(* PLC project Unnamed, Unknown Unnamed 1 *)
(* stored: creationDateTime 2024-11-21T00:40:53, modificationDateTime 2024-12-05T23:30:09 *)

(* LED *)
PROGRAM HelloWorld
  VAR
    Set : BOOL;
    Reset : BOOL;
    Hello_World : BOOL;
    Select : INT;
    Mode_1 : BOOL;
    Mode_2 : BOOL;
    Mode_3 : BOOL;
    Mode_4 : BOOL;
    LED : BOOL;
    LED0 : BOOL;
    R_TRIG0 : R_TRIG;
    F_TRIG0 : F_TRIG;
  END_VAR
  VAR  (* added by the conversion: wires and edge detectors of the diagram *)
    _MOVE27_ENO : BOOL;
    _MOVE27_OUT : INT;
  END_VAR

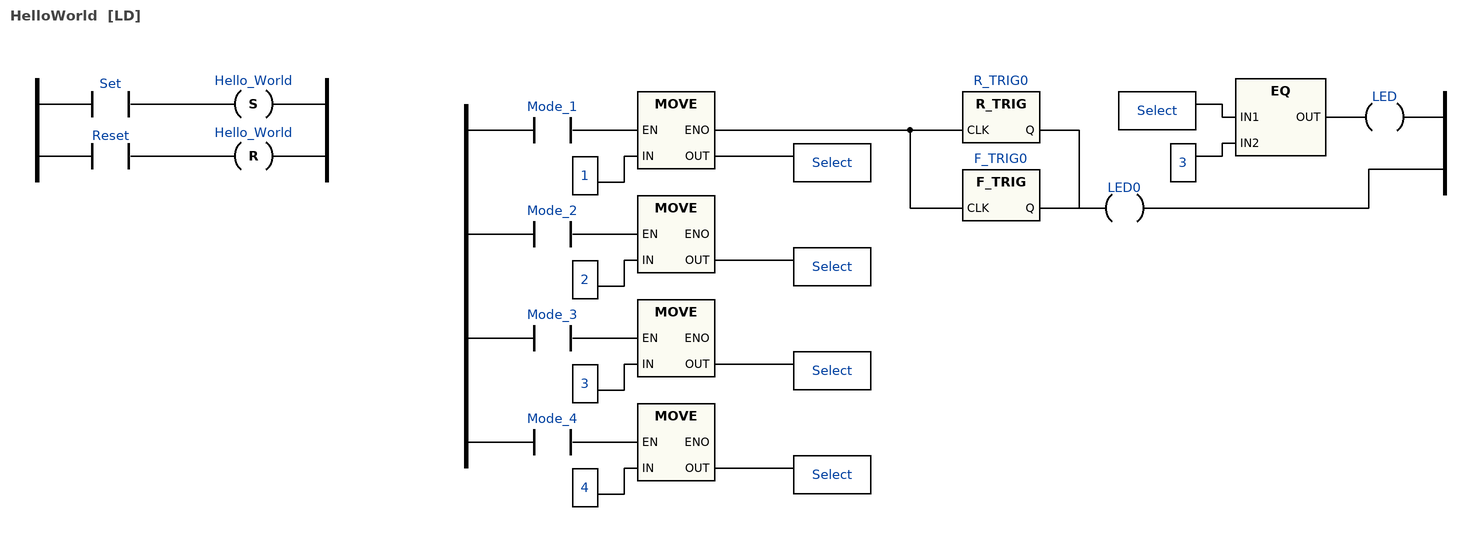
(* LD diagram, written out as Structured Text *)
IF Set THEN Hello_World := TRUE; END_IF;
IF Reset THEN Hello_World := FALSE; END_IF;
_MOVE27_OUT := MOVE(EN := Mode_1, IN := 1, ENO => _MOVE27_ENO);
IF _MOVE27_ENO THEN Select := _MOVE27_OUT; END_IF;
IF Mode_2 THEN Select := 2; END_IF;
IF Mode_3 THEN Select := 3; END_IF;
IF Mode_4 THEN Select := 4; END_IF;
LED := Select = 3;
R_TRIG0(CLK := _MOVE27_ENO);
F_TRIG0(CLK := _MOVE27_ENO);
LED0 := R_TRIG0.Q OR F_TRIG0.Q;
END_PROGRAM

CONFIGURATION Config0
  RESOURCE Res0 ON PLC
    TASK task0(INTERVAL := T#20ms, PRIORITY := 0);
    PROGRAM instance0 WITH task0 : HelloWorld;
  END_RESOURCE
END_CONFIGURATION
